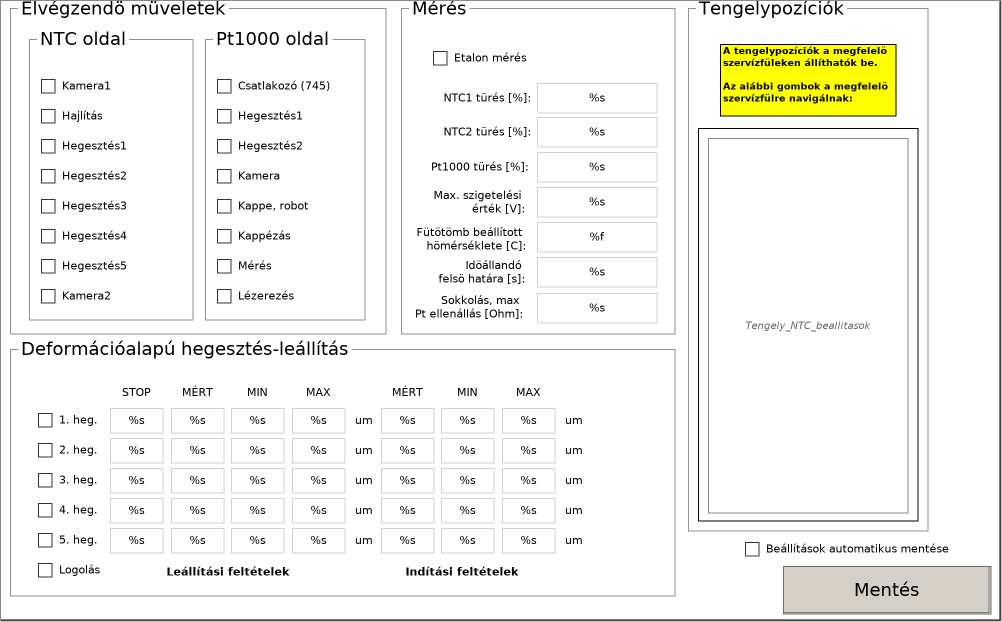
VISUALIZATION Beallitasok  // 1002x622
    Rectangle (0,0 1000x620)
    GroupBox (10,0 376x334), "Elvégzendö müveletek"
        GroupBox (19,31 164x289), "NTC oldal"
            Checkbox (10,70 140x30), "Hajlítás", variable: GVL.bHajlitasBe, input disabled if: AUTOMATA.bFolyamatBeallitas1Tiltva
            Checkbox (10,100 140x30), "Hegesztés1", variable: GVL.bHegesztes1Be, input disabled if: AUTOMATA.bFolyamatBeallitas1Tiltva
            Checkbox (10,130 140x30), "Hegesztés2", variable: GVL.bHegesztes2Be, input disabled if: AUTOMATA.bFolyamatBeallitas1Tiltva
            Checkbox (10,160 140x30), "Hegesztés3", variable: GVL.bHegesztes3Be, input disabled if: AUTOMATA.bFolyamatBeallitas1Tiltva
            Checkbox (10,190 140x30), "Hegesztés4", variable: GVL.bHegesztes4Be, input disabled if: AUTOMATA.bFolyamatBeallitas1Tiltva
            Checkbox (10,220 140x30), "Hegesztés5", variable: GVL.bHegesztes5Be, input disabled if: AUTOMATA.bFolyamatBeallitas1Tiltva
            Checkbox (10,40 140x30), "Kamera1", variable: GVL.bKameraBe, input disabled if: AUTOMATA.bFolyamatBeallitas1Tiltva
            Checkbox (10,250 140x30), "Kamera2", variable: GVL.bKameraVegBe, input disabled if: AUTOMATA.bFolyamatBeallitas1Tiltva
        GroupBox (195,31 160x289), "Pt1000 oldal"
            Checkbox (10,250 140x30), "Lézerezés", variable: GVL.bJelolesBe, input disabled if: AUTOMATA.bFolyamatBeallitas2Tiltva
            Checkbox (10,70 140x30), "Hegesztés1", variable: GVL.bHegesztes6Be, input disabled if: AUTOMATA.bFolyamatBeallitas2Tiltva
            Checkbox (10,100 140x30), "Hegesztés2", variable: GVL.bHegesztes7Be, input disabled if: AUTOMATA.bFolyamatBeallitas2Tiltva
            Checkbox (10,160 140x30), "Kappe, robot", variable: GVL.bRobotKappeBe, input disabled if: AUTOMATA.bFolyamatBeallitas2Tiltva
            Checkbox (10,190 140x30), "Kappézás", variable: GVL.bKappeBe, input disabled if: AUTOMATA.bFolyamatBeallitas2Tiltva
            Checkbox (10,220 140x30), "Mérés", variable: GVL.bMeresBe, input disabled if: AUTOMATA.bFolyamatBeallitas2Tiltva
            Checkbox (10,130 140x30), "Kamera", variable: GVL.bPtKameraBe, input disabled if: AUTOMATA.bFolyamatBeallitas2Tiltva AND TRUE
            Checkbox (10,40 140x30), "Csatlakozó (745)", variable: GVL.bHimbaBe, input disabled if: AUTOMATA.bFolyamatBeallitas2Tiltva AND (GVL.iSelectedProductType<=8)
    GroupBox (401,0 274x334), "Mérés"
        Checkbox (30,43 116x30), "Etalon mérés", variable: GVL.bEtalonOn
        Textfield (136,83 120x30), "%s", text variable: GVL.rNTCDev
            OnMouseClick: write the text variable via VisuDialogs.Numpad, min 0, max 30
        Label (42,83 89x30), "NTC1 türés [%]:"
        Textfield (136,187 120x30), "%s", text variable: GVL.rISOL_MAX
            OnMouseUp: write the text variable via VisuDialogs.Numpad, min 0, max 2
        Label (34,187 93x30), "Max. szigetelési érték [V]:"
        Textfield (136,222 120x30), "%f", text variable: GVL.rTempMax
            OnMouseClick: write the text variable via VisuDialogs.Numpad, min 0, max 400
        Label (54,257 73x30), "Idöállandó felsö határa [s]:"
        Textfield (136,257 120x30), "%s", text variable: GVL.rIdoallandoMax
            OnMouseClick: write the text variable via VisuDialogs.Numpad, min 0, max 8
        Textfield (136,152 120x30), "%s", text variable: GVL.rPtDev
            OnMouseClick: write the text variable via VisuDialogs.Numpad, min 0, max 15
        Label (27,152 104x30), "Pt1000 türés [%]:"
        Textfield (136,293 120x30), "%s", text variable: GVL.PTRES_SOKK_MAX
            OnMouseClick: write the text variable via VisuDialogs.Numpad, min 0, max 3000
        Label (22,222 106x34), "Fütötömb beállított hömérséklete [C]:"
        Label (11,292 114x30), "Sokkolás, max Pt ellenállás [Ohm]:"
        Label (42,117 89x30), "NTC2 türés [%]:"
    GroupBox (688,0 240x531), "Tengelypozíciók"
        Rectangle (32,44 176x72), "A tengelypozíciók a megfelelö szervízfüleken állíthatók be. Az alábbi gombok a megfelelö szervízfülre navigálnak:"
        Rectangle (10,128 220x393)
        TabControl (20,138 200x375)
            shows Tengely_NTC_beallitasok()
            shows Tengely_Pt1000_beallitasok()
            [0]: TabTitle=NTC oldal
            [1]: TabTitle=Pt1000 oldal
    GroupBox (10,341 665x255), "Deformációalapú hegesztés-leállítás"
        Checkbox (26,154 75x30), "4. heg.", variable: GVL.bAutomaticWeldingStop4
        Checkbox (26,184 75x30), "5. heg.", variable: GVL.bAutomaticWeldingStop5
        Checkbox (26,124 75x30), "3. heg.", variable: GVL.bAutomaticWeldingStop3
        Checkbox (26,94 75x30), "2. heg.", variable: GVL.bAutomaticWeldingStop2
        Checkbox (26,64 75x30), "1. heg.", variable: GVL.bAutomaticWeldingStop1
        Textfield (100,187 53x25), "%s", text variable: GVL.nWeldingStopDistance5
            OnMouseClick: write the text variable via VisuDialogs.Numpad, min 0, max 1000
        Textfield (100,157 53x25), "%s", text variable: GVL.nWeldingStopDistance4
            OnMouseClick: write the text variable via VisuDialogs.Numpad, min 0, max 1000
        Textfield (100,127 53x25), "%s", text variable: GVL.nWeldingStopDistance3
            OnMouseClick: write the text variable via VisuDialogs.Numpad, min 0, max 1000
        Textfield (100,97 53x25), "%s", text variable: GVL.nWeldingStopDistance2
            OnMouseClick: write the text variable via VisuDialogs.Numpad, min 0, max 1000
        Textfield (100,67 53x25), "%s", text variable: GVL.nWeldingStopDistance1
            OnMouseClick: write the text variable via VisuDialogs.Numpad, min 0, max 1000
        Textfield (161,67 53x25), "%s", text variable: GVL.nWeldingDeformation1
        Textfield (161,97 53x25), "%s", text variable: GVL.nWeldingDeformation2
        Textfield (161,127 53x25), "%s", text variable: GVL.nWeldingDeformation3
        Textfield (161,157 53x25), "%s", text variable: GVL.nWeldingDeformation4
        Textfield (161,187 53x25), "%s", text variable: GVL.nWeldingDeformation5
        Label (104,39 45x25), "STOP"
        Label (165,39 45x25), "MÉRT"
        Checkbox (26,214 87x30), "Logolás", variable: GVL.bWeldingLog
        Label (342,67 25x25), "um"
        Label (342,97 25x25), "um"
        Label (342,127 25x25), "um"
        Label (342,157 25x25), "um"
        Label (342,187 25x25), "um"
        Textfield (221,67 53x25), "%s", text variable: GVL.nWeldingDistanceMin1
            OnMouseClick: write the text variable via VisuDialogs.Numpad, min 0, max 2000
        Label (225,39 45x25), "MIN"
        Label (143,216 150x30), "Leállítási feltételek"
        Label (377,216 150x30), "Indítási feltételek"
        Textfield (371,97 53x25), "%s", text variable: GVL.ulWeldingStartDistance2
        Textfield (371,127 53x25), "%s", text variable: GVL.ulWeldingStartDistance3
        Textfield (371,187 53x25), "%s", text variable: GVL.ulWeldingStartDistance5
    Checkbox (743,534 223x30), "Beállítások automatikus mentése", variable: GVL.bSettingsAutoSave
    Button (783,566 208x48), "Mentés"
        OnMouseClick: execute { MAIN.iStateS:=3; }
    Textfield (231,528 53x25), "%s", text variable: GVL.nWeldingDistanceMin5
        OnMouseClick: write the text variable via VisuDialogs.Numpad, min 0, max 2000
    Textfield (231,498 53x25), "%s", text variable: GVL.nWeldingDistanceMin4
        OnMouseClick: write the text variable via VisuDialogs.Numpad, min 0, max 2000
    Textfield (231,468 53x25), "%s", text variable: GVL.nWeldingDistanceMin3
        OnMouseClick: write the text variable via VisuDialogs.Numpad, min 0, max 2000
    Textfield (231,438 53x25), "%s", text variable: GVL.nWeldingDistanceMin2
        OnMouseClick: write the text variable via VisuDialogs.Numpad, min 0, max 2000
    Textfield (292,408 53x25), "%s", text variable: GVL.nWeldingDistanceMax1
        OnMouseClick: write the text variable via VisuDialogs.Numpad, min 0, max 2000
    Textfield (292,438 53x25), "%s", text variable: GVL.nWeldingDistanceMax2
        OnMouseClick: write the text variable via VisuDialogs.Numpad, min 0, max 2000
    Textfield (292,468 53x25), "%s", text variable: GVL.nWeldingDistanceMax3
        OnMouseClick: write the text variable via VisuDialogs.Numpad, min 0, max 2000
    Textfield (292,498 53x25), "%s", text variable: GVL.nWeldingDistanceMax4
        OnMouseClick: write the text variable via VisuDialogs.Numpad, min 0, max 2000
    Textfield (292,528 53x25), "%s", text variable: GVL.nWeldingDistanceMax5
        OnMouseClick: write the text variable via VisuDialogs.Numpad, min 0, max 2000
    Label (296,380 45x25), "MAX"
    Textfield (381,408 53x25), "%s", text variable: GVL.ulWeldingStartDistance1
    Textfield (381,498 53x25), "%s", text variable: GVL.ulWeldingStartDistance4
    Label (385,380 45x25), "MÉRT"
    Label (562,408 25x25), "um"
    Label (562,438 25x25), "um"
    Label (562,468 25x25), "um"
    Label (562,498 25x25), "um"
    Label (562,528 25x25), "um"
    Textfield (441,408 53x25), "%s", text variable: GVL.nWeldingDistanceStartMin1
        OnMouseClick: write the text variable via VisuDialogs.Numpad, min 0, max 200000
    Label (445,380 45x25), "MIN"
    Textfield (441,528 53x25), "%s", text variable: GVL.nWeldingDistanceStartMin5
        OnMouseClick: write the text variable via VisuDialogs.Numpad, min 0, max 200000
    Textfield (441,498 53x25), "%s", text variable: GVL.nWeldingDistanceStartMin4
        OnMouseClick: write the text variable via VisuDialogs.Numpad, min 0, max 200000
    Textfield (441,468 53x25), "%s", text variable: GVL.nWeldingDistanceStartMin3
        OnMouseClick: write the text variable via VisuDialogs.Numpad, min 0, max 200000
    Textfield (441,438 53x25), "%s", text variable: GVL.nWeldingDistanceStartMin2
        OnMouseClick: write the text variable via VisuDialogs.Numpad, min 0, max 200000
    Textfield (502,408 53x25), "%s", text variable: GVL.nWeldingDistanceStartMax1
        OnMouseClick: write the text variable via VisuDialogs.Numpad, min 0, max 210000
    Textfield (502,438 53x25), "%s", text variable: GVL.nWeldingDistanceStartMax2
        OnMouseClick: write the text variable via VisuDialogs.Numpad, min 0, max 210000
    Textfield (502,468 53x25), "%s", text variable: GVL.nWeldingDistanceStartMax3
        OnMouseClick: write the text variable via VisuDialogs.Numpad, min 0, max 210000
    Textfield (502,498 53x25), "%s", text variable: GVL.nWeldingDistanceStartMax4
        OnMouseClick: write the text variable via VisuDialogs.Numpad, min 0, max 210000
    Textfield (502,528 53x25), "%s", text variable: GVL.nWeldingDistanceStartMax5
        OnMouseClick: write the text variable via VisuDialogs.Numpad, min 0, max 210000
    Label (506,380 45x25), "MAX"
    Textfield (537,117 120x30), "%s", text variable: GVL.rNTC2Dev
        OnMouseClick: write the text variable via VisuDialogs.Numpad, min 0, max 30
END_VISUALIZATION

(* stored: Version 1.1.0.1, ProductVersion 3.1.4024.11
   Visu Beallitasok: Id {9bf3f38c-3524-4dc0-81f0-f6c760b4e396} *)
